(* PLC project Generated.project, CODESYS CODESYS V3.5 SP19 Patch 1 *)
(* stored: creationDateTime 2026-09-21T00:59:23.792961, modificationDateTime 2026-09-21T00:59:23.792961 *)

(* ======================================================================= 🔄 ST_ChainCycleSemiAuto — Diagnostic chronologique Séquenceur Semi-Auto ─────────────────────────────────────────────────────────────── 🎯 Rôle : Vue dépannage / Watch CODESYS pour le cycle semi-automatique 📄 Doc métier : DOC/AF/AF_Partie-14_Fonction_Troubleshooting/FB_TroubleshootingView_v1.2.md 🔒 Sécurité : 100% lecture seule / diagnostic d'observation ======================================================================= *)
TYPE ST_ChainCycleSemiAuto : STRUCT
  Idx101_ModeSemiAutoActive : BOOL;  (* 🚦 1. Conditions d'engagement et autorisations 1 = Mode arbitré SEMI_AUTO actif | 0 = Autre mode *)
  Idx102_PowerAndSafetyOk : BOOL;  (* 1 = Chaîne de sécurité OK (PowerContactorEngaged) *)
  Idx103_HeartbeatIhmOk : BOOL;  (* 1 = Liaison IHM<->PLC valide *)
  Idx104_DeadmanArmed : BOOL;  (* 1 = Bouton homme-mort armé (fenêtre 3s active) *)
  Idx105_MancheDeflechi : BOOL;  (* 1 = Permis mouvement armé (manche hors zone neutre) *)
  Idx106_HomedM1M2 : BOOL;  (* 1 = Codeurs treuils M1 et M2 référencés *)
  Idx107_StartCycleRequest : BOOL;  (* 1 = Demande Start reçue (IHM) *)
  Idx108_AbortCycleRequest : BOOL;  (* 1 = Demande Abort reçue (IHM) *)
  Idx201_Ready : BOOL;  (* 🔄 2. État du Séquenceur 1 = Séquenceur prêt à démarrer *)
  Idx202_Busy : BOOL;  (* 1 = Cycle en cours d'exécution *)
  Idx203_Done : BOOL;  (* 1 = Cycle terminé avec succès *)
  Idx204_Error : BOOL;  (* 1 = Défaut vue LIVE (retombe seul avec la cause) *)
  Idx205_ErrorId : WORD;  (* Code d'erreur interne FB_Cycle *)
  Idx217_FaultLatched : BOOL;  (* 1 = Défaut vue LATCHÉE (bloque AX0->AX1 même si Idx204=0, exige Reset conscient) *)
  Idx218_FaultLatchedId : WORD;  (* Bitfield fige a l'apparition du defaut latche *)
  Idx219_CycleChecksInhibited : BOOL;  (* 1 = controles procede inhibes, protections actives *)
  Idx220_IgnoredCycleCheckId : WORD;  (* Causes procede actives mais ignorees *)
  Idx222_ForceStepResult : STRING(120);  (* ⚠️ Idx221 (ForceStepPrepared) SUPPRIME par T358 : le mecanisme a deux temps du forcage de step n'existe plus (saut immediat sans preparation). L'index reste VACANT pour ne renumeroter aucun tag IHM de la chaine de depannage. Motif de rejet de la derniere consigne de forcage (T358) *)
  Idx206_Step : E_AutoCycleStep;  (* Étape courante (X0 à X13 + AX_STAB) *)
  Idx207_StepStr : STRING(80);  (* Libellé explicite de l'étape *)
  Idx208_StepAtError : E_AutoCycleStep;  (* Étape mémorisée lors du dernier défaut *)
  Idx209_WaitingForOperator : BOOL;  (* 1 = En attente d'une action humaine *)
  Idx210_WaitingForProcess : BOOL;  (* 1 = En attente d'une condition physique/procédé *)
  Idx211_OperatorActionId : WORD;  (* Identifiant numérique de l'action attendue *)
  Idx212_OperatorAction : STRING(120);  (* Description explicite de l'action/attente *)
  Idx213_ExpectedAxis : E_OperatorAxis;  (* Organe attendu (NONE, JOYSTICK_X, JOYSTICK_Y, BUTTON) *)
  Idx214_ExpectedDirection : INT;  (* Sens attendu (-1, 0, +1) *)
  Idx215_WaitingResume : BOOL;  (* 1 = En pause suite à bascule de mode (attente StartCycle) *)
  Idx216_PausedState : E_AutoCycleStep;  (* Étape mémorisée prête pour reprise *)
  Idx301_TargetPosition : INT;  (* 🎯 3. Consignes & Feedbacks Opérationnels Cible translation sélectionnée (1=Trémie, 3=P1) *)
  Idx302_TargetDepth_M : REAL;  (* Profondeur de consigne (m) *)
  Idx303_KoboldBottomTouch : BOOL;  (* 1 = Détection contact fond Kobold *)
  Idx304_SpeedMismatchActive : BOOL;  (* 1 = Alerte écart de vitesse M1/M2 active *)
  Idx305_LimitLegalReached : BOOL;  (* 1 = Limite légale atteinte (descente bloquée) *)
  Idx306_WinchSyncError : BOOL;  (* 1 = Erreur de synchronisme M1/M2 *)
  Idx307_M1SpeedStepApplied : INT;  (* Palier vitesse applique M1 (0..5, causes 8/9) *)
  Idx308_M2SpeedStepApplied : INT;  (* Palier vitesse applique M2 (0..5, causes 8/9) *)
  Idx309_AutoDiveM2Step5Active : BOOL;  (* 1 = Essai T291-A actif (M2 cible palier 5 en plongee) *)
  Idx310_M1SpeedStepAtFault : INT;  (* Palier M1 applique, fige au moment du defaut (0..5) *)
  Idx311_M2SpeedStepAtFault : INT;  (* Palier M2 applique, fige au moment du defaut (0..5) *)
END_STRUCT;
END_TYPE

(* values of E_AutoCycleStep: AX0_REPOS: Repos / park : toutes commandes 0, etat neutre - etape initiale pure; AX1_INIT: Verif CONDITIONS INITIALES (Homed M1/M2, treuils FDC haut, M3 pas a droite de P1) - aucun mouvement, aucun referencement; AX2_TRANSLATE_P1: Translation vers P1 : joystick vers la droite, le cycle n'emet aucune commande M3 ; surveillance treuils au FDC haut; AX3_OPEN_BUCKET: Ouverture benne jusqu'au FDC logiciel benne ouverte --- DIVING (5 steps + retry) ---; AX4_DESCEND_DIVING: Plongee couplee benne ouverte palier 4 jusqu'a l'altimetrie de lancement (DiveStartMin_M) - Kobold PAS enclenche; AX5_KOBOLD_INIT: Activation contacteur Kobold << au vol >>, verif retour contacteur, descente palier 4 maintenue; AX6_SEARCH_IMMERSION: Recherche entree dans l'eau : attente front DI Kobold 0->1, descente palier 4 maintenue; AX7_SEARCH_BOTTOM: Recherche du fond : attente front DI Kobold 1->0, descente palier 4 maintenue; AX8_BOTTOM_CONFIRMED: Fond confirme : coupure instantanee treuils, set bit fond, TouchPositionM / RaiseTargetM --- EXTRACTION (4 steps) ---; AX9_RAISE_OFF_BOTTOM: Montee synchronisee : retendre les cables ; selecteur couplage BOTH/M1/M2 accessible; AX10_CLOSE_BUCKET: Fermeture benne, treuils explicitement 0; AX11_CTRL_ASCENT: Montee controle palier max reglable [1..2] + surveillance ecart vitesse M1/M2 ; benne mal fermee autorisee; AX12_LOADED_ASCENT: Montee en charge : palier 4 si benne fermee, palier 1 si mal fermee ; pas de ralenti 1 m avant top --- DECHARGE (6 steps) ---; AX13_DRAIN_PAUSE: Egouttage temporise - duree reglable IHM + bypass immediat; AX14_TRANSLATE_DUMP: Translation vers tremie (depart P1) + avertissements IHM; AX15A_DUMP_ARRIVE: Arrivee tremie : treuils a l'arret, attente geste operateur; AX15B_DUMP_OPEN: Vidage : ouverture benne au-dessus de la tremie, LES DEUX treuils a l'arret; AX15C_DUMP_REPOSITION: Repositionnement couple M1+M2 (option IHM maintenue), retour AX15B au relachement; AX18_DONE_SYNC: Fin de passe : compteur vidages + duree cycle ; msg << aller en P1 >> ; rebouclage direct sur AX2 --- STEPS SPECIAUX ---; AX_STAB: Repli defaut / stabilisation - pas une erreur; AX_DIVING_RETRY: Reprise diving : remontee assistee palier lent jusqu'au FDC haut puis retour AX4 ; sur erreur Kobold / joystick relache / palier <> 4 en AX5..AX7; AX3_WAIT_DIVE_START: Transition benne->plongee : sorties neutres jusqu'a l'arret mecanique confirme M1/M2, joystick pousse maintenu; AX10B_RACCORDEMENT_P1: Raccordement continu P1 fermeture benne -> montee controlee *)

{attribute 'qualified_only'}
{attribute 'strict'}
TYPE E_AutoCycleStep : (AX0_REPOS := 0, AX1_INIT := 1, AX2_TRANSLATE_P1 := 2, AX3_OPEN_BUCKET := 3, AX4_DESCEND_DIVING := 4, AX5_KOBOLD_INIT := 5, AX6_SEARCH_IMMERSION := 6, AX7_SEARCH_BOTTOM := 7, AX8_BOTTOM_CONFIRMED := 8, AX9_RAISE_OFF_BOTTOM := 9, AX10_CLOSE_BUCKET := 10, AX11_CTRL_ASCENT := 11, AX12_LOADED_ASCENT := 12, AX13_DRAIN_PAUSE := 13, AX14_TRANSLATE_DUMP := 14, AX15A_DUMP_ARRIVE := 15, AX15B_DUMP_OPEN := 16, AX15C_DUMP_REPOSITION := 17, AX18_DONE_SYNC := 18, AX_STAB := 19, AX_DIVING_RETRY := 20, AX3_WAIT_DIVE_START := 21, AX10B_RACCORDEMENT_P1 := 22);
END_TYPE

(* values of E_OperatorAxis: NONE: Aucun axe attendu (étape automatique ou arrêt); JOYSTICK_X: Axe X translation attendu; JOYSTICK_Y: Axe Y treuils / plongée attendu; BUTTON: Action bouton attendue (ex: validation, homing) *)

{attribute 'qualified_only'}
{attribute 'strict'}
TYPE E_OperatorAxis : (NONE := 0, JOYSTICK_X := 1, JOYSTICK_Y := 2, BUTTON := 3);
END_TYPE
